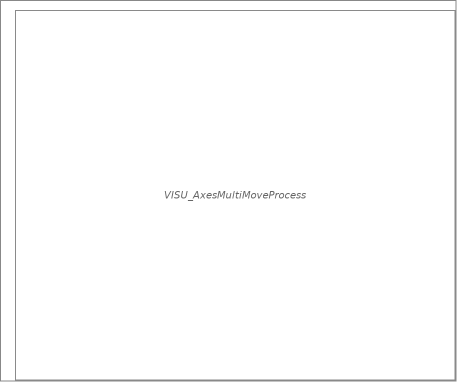
VISUALIZATION VISU_AxesManual_MoveAbsolute  // 457x382
VAR_IN_OUT
	ref : Axes;
    widget : AxesManualMoveAbsoluteWidget;
END_VAR
    Frame (15,10 440x370)
        shows VISU_AxesMultiMoveProcess(ref := ref.processes.moveAbsolute, widget := widget.moveAbsolute)
END_VISUALIZATION

(* stored: Version 1.1.0.1, ProductVersion 3.1.4019.2
   Visu VISU_AxesManual_MoveAbsolute: Id {4ac98481-bfd4-4c36-b15d-299c0648cb9c} *)
